FUNCTION_BLOCK SP_MoveArm (* MoveArm parameters (Angle [deg] 0.0..180.0, default 120.0; Settle [s] 0.0..5.0, default 2.0): OPC UA IDs, range check and latching *)
  (* Standard: 61499-2 *)
  (* Version 0.1, 2026-09-28, Project contributors, AAU Smart Production Lab *)
  PACKAGE stoppering;
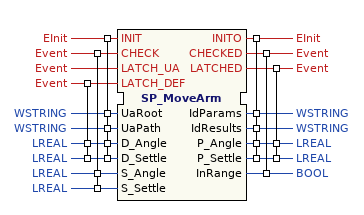
  EVENT_INPUT
    INIT : EInit WITH UaRoot, UaPath, D_Angle, D_Settle;
    CHECK WITH S_Angle, S_Settle;
    LATCH_UA;
    LATCH_DEF WITH D_Angle, D_Settle;
  END_EVENT
  EVENT_OUTPUT
    INITO : EInit WITH IdParams, IdResults, P_Angle, P_Settle;
    CHECKED WITH InRange;
    LATCHED WITH P_Angle, P_Settle;
  END_EVENT
  VAR_INPUT
    UaRoot : WSTRING;
    UaPath : WSTRING;
    D_Angle : LREAL;
    D_Settle : LREAL;
    S_Angle : LREAL;
    S_Settle : LREAL;
  END_VAR
  VAR_OUTPUT
    IdParams : WSTRING;
    IdResults : WSTRING;
    P_Angle : LREAL;
    P_Settle : LREAL;
    InRange : BOOL;
  END_VAR
  EC_STATES
    INIT : INIT -> INITO;
    CHECK : CHECK -> CHECKED;
    LATCH_UA : LATCH_UA -> LATCHED;
    LATCH_DEF : LATCH_DEF -> LATCHED;
  END_STATES
  ALGORITHM INIT IN ST:
IdParams := CONCAT(CONCAT(CONCAT(CONCAT(CONCAT("opc_ua[WRITE;", CONCAT(UaRoot, UaPath)), "/Parameters/Angle;"), CONCAT(UaRoot, UaPath)), "/Parameters/Settle"), "]");
IdResults := "";
P_Angle := D_Angle;
P_Settle := D_Settle;
  END_ALGORITHM
  ALGORITHM CHECK IN ST:
InRange := (S_Angle >= 0.0) AND (S_Settle >= 0.0) AND (S_Angle <= 180.0) AND (S_Settle <= 5.0);
  END_ALGORITHM
  ALGORITHM LATCH_UA IN ST:
P_Angle := S_Angle;
P_Settle := S_Settle;
  END_ALGORITHM
  ALGORITHM LATCH_DEF IN ST:
P_Angle := D_Angle;
P_Settle := D_Settle;
  END_ALGORITHM
END_FUNCTION_BLOCK
